// TIA Portal V17 export
// export: Created 2023-12-22T15:04:45.1327482Z, ExportSetting WithDefaults, DisplayName Totally Integrated Automation Portal, DisplayVersion V17, DisplayName TIA Portal Openness, DisplayVersion V17, DisplayName TIA Portal Version Control Interface, DisplayVersion V17, DisplayName STEP 7 Professional, DisplayVersion V17, DisplayName STEP 7 Safety, DisplayVersion V17, DisplayName WinCC Advanced, DisplayVersion V17
DATA_BLOCK "Comm_SKD1_DB"   // DB10
VERSION : 0.1
// stored: AutoNumber false, DBAccessibleFromOPCUA true, InstanceOfName Comm_SKD1, InstanceOfType FB
"Comm_SKD1"
   // VAR RETAIN
   //    From_SKD1 : Struct
   //       watchdog : Int;
   //       LE_1 : Int;
   //       LE_2 : Int;
   //       LE_3 : Int;
   //       LE_4 : Int;
   //       SP_FE : Int;
   //       SP_M : Int;
   //       CMD : Struct
   //          REQ : Bool;
   //          Reset : Bool;
   //          Hand : Bool;
   //          Start_M : Bool;
   //       END_STRUCT;
   //       Valves : Struct
   //          ID : Int;
   //          Local : Array[0..15] of Bool;
   //          Mode : Array[1..10] of Int;
   //          Status : Array[1..10] of Int;
   //       END_STRUCT;
   //    END_STRUCT;
   //    To_SKD1 : Struct
   //       watchdog : Int;
   //       LE_SKV : Int;
   //       res_h : DInt;
   //       LE : Int;
   //       TE : Int;
   //       PE_1 : Int;
   //       PE_2 : Int;
   //       PE_3 : Int;
   //       PE_4 : Int;
   //       FE : Int;
   //       C : Int;
   //       Status : Int;
   //       STATE : Struct
   //          Ready : Bool;
   //          Local : Bool;
   //          Warning : Bool;
   //          Alarm : Bool;
   //          LS : Bool;
   //          Lock : Bool;
   //       END_STRUCT;
   //       Valves : Struct
   //          ID : Int;
   //          REQ : Array[0..15] of Bool;
   //       END_STRUCT;
   //    END_STRUCT;
   //    Alarm : Struct
   //       Link : Bool;
   //    END_STRUCT;
   //    watchdog_control : Int;
   //    ID : Int;
   //    LE_1 : Real;
   //    LE_2 : Real;
   //    LE_3 : Real;
   //    LE_4 : Real;
   //    Valve_Name { S7_SetPoint := 'True'} : Array[1..10] of String[4];
   //    Clock : Array[0..10] of "Time_S";
   // END_VAR
BEGIN
   Valve_Name[1..10] := '';
END_DATA_BLOCK
